RoboDK station: main_station.rdk

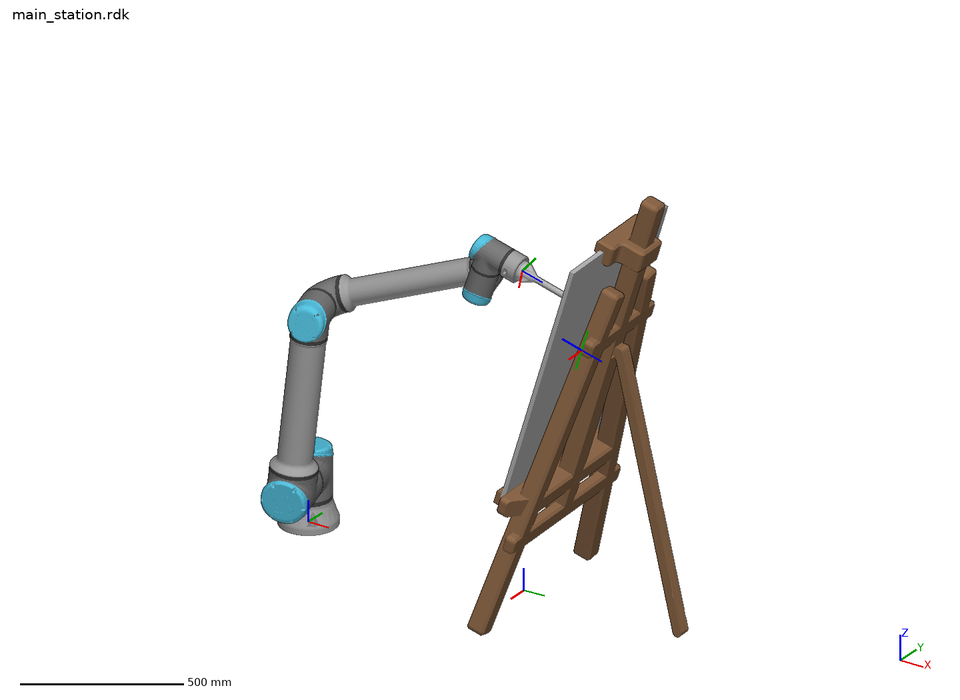
[picture v0: the station drawn from its stored meshes, robots at their saved joint values, targets as dots, program paths as lines]
Station main_station (saved by RoboDK 5.6.7). Poses are relative to the parent item; angles as X-Y-Z fixed-axis rotations.
Station parameters (name, value as stored): LIN64
  - frame UR10e Base at (0, 0, 0) mm
    - robot UR10e: 6 axes, payload 10 kg, reach 1300 mm, repeatability 0.05 mm, weight 28.9 kg
        modified DH rows (alpha deg, a mm, theta deg, d mm): 0, 0, 0, 180.7; 90, 0, 180, 0; 0, 612.6, 0, 0; 0, 571.335, 0, 174.15; -90, 0, 0, 119.85; 90, 0, 180, 116.55
        joint limits [-360, -360, -360, -360, -360, -360] to [360, 360, 360, 360, 360, 360]; home [0, -90, -90, 0, 90, 0]; saved at [17.363, -95.973, -65.265, -35.905, 76.874, 106.533]
      - frame flange at (0, 0, 0) mm
        - object pen_holder at (26.63, 0, 42.81) mm, rotated rx 180 ry 0 rz 180 deg, size 63 x 63 x 153.3 mm, geometry from penholder_Chamfer003.stl
      - tool marker, TCP at (0, 0, 160) mm
    - frame canvas at (1017.6, 1.12, 865.8) mm, rotated rx -106.68 ry 0 rz -86.35 deg
      - object canvas at (0, 0, 8.06) mm, rotated rx 90 ry 0 rz 0 deg, size 551.3 x 14.9 x 864.2 mm, geometry from canvas.stl
      - frame canvas_offset at (0, 0, 0) mm, rotated rx -180 ry 0 rz 0 deg
  - frame easel at (809.92, -12.12, 0) mm, rotated rx 0 ry 0 rz -86.35 deg
    - object EASEL SMALL at (-1879.48, -1290.24, -11.21) mm, size 684 x 573 x 1450.9 mm, geometry from EASEL SMALL.stl
